{attribute addProperty BoxType "EK1122-0000-0018"}
{attribute addProperty Id "Beckhoff_EPP3xxxsub_EK1100EK1100_179A0949162A_0001_EPP3174_0002_0016EPP3174_B7B5302521026.25A_0002_EPP3174_0002_0017EPP3174_B7B5302521026.25A_0003_EPP3174_0002_0018EPP3174_B7B5302521026.25A_0004_EPP3184_0002_0016EPP3184_6082EBFD21026.25A_0005_EPP3184_0002_0017EPP3184_6082EBFD21026.25A_0006_EPP3184_0002_0018EPP3184_6082EBFD21026.25A_0007_EPP3184_0002_0019EPP3184_B7B5302521026.25A_0008_EPP3204_0002_0016EPP3204_72ABB95437847.25A_0009_EPP3204_0002_0017EPP3204_C91659E221026.25A_0010_EPP3204_0002_0018EPP3204_C91659E221026.25A_0011_EPP3204_0002_0019EPP3204_C91659E221026.25A_0012_EPP3314_0002_0016EPP3314_A69716D721026.25A_0013_EPP3314_0002_0017EPP3314_A69716D721026.25A_0014_EPP3314_0002_0018EPP3314_A69716D721026.25A_0015_EPP3632_0001_0016EPP3632_A724E07457872.25A_0016_EPP3632_0001_0017EPP3632_A724E07457872.25A_0017_EPP3744_0041_0016EPP3744_99A8040A38648.25A_0018_EPP3744_0041_0017EPP3744_99A8040A38648.25A_0019_EPP3744_0041_0018EPP3744_99A8040A38648.25A_0020_EPP3744_1041_0016EPP3744_99A8040A38648.25A_0021_EPP3744_1041_0017EPP3744_99A8040A38648.25A_0022_EPP3744_1041_0018EPP3744_99A8040A38648.25A_0023_EPP3744_1041_0019EPP3744_99A8040A38648.25A_0024_EPP3744_1041_0020EPP3744_99A8040A38648.25A_0025_EPP3752_0000_0017EPP3752_639ED5F327434.25"}
{attribute addProperty CRC "2472904185"}
{attribute addProperty SizeInBites "7642"}
{attribute addProperty SizeInBytes "955.25"}
TYPE Beckhoff_EPP3xxxEK1122_936585F9 EXTENDS EK1122_179A0949 :
STRUCT
	{attribute addProperty Name "Beckhoff_EPP3xxxsub_EK1100"}
	Beckhoff_EPP3xxxsub_EK1100 : EK1100_179A0949;
	{attribute addProperty Name "A_0001_EPP3174_0002_0016"}
	A_0001_EPP3174_0002_0016 : EPP3174_B7B53025;
	{attribute addProperty Name "A_0002_EPP3174_0002_0017"}
	A_0002_EPP3174_0002_0017 : EPP3174_B7B53025;
	{attribute addProperty Name "A_0003_EPP3174_0002_0018"}
	A_0003_EPP3174_0002_0018 : EPP3174_B7B53025;
	{attribute addProperty Name "A_0004_EPP3184_0002_0016"}
	A_0004_EPP3184_0002_0016 : EPP3184_6082EBFD;
	{attribute addProperty Name "A_0005_EPP3184_0002_0017"}
	A_0005_EPP3184_0002_0017 : EPP3184_6082EBFD;
	{attribute addProperty Name "A_0006_EPP3184_0002_0018"}
	A_0006_EPP3184_0002_0018 : EPP3184_6082EBFD;
	{attribute addProperty Name "A_0007_EPP3184_0002_0019"}
	A_0007_EPP3184_0002_0019 : EPP3184_B7B53025;
	{attribute addProperty Name "A_0008_EPP3204_0002_0016"}
	A_0008_EPP3204_0002_0016 : EPP3204_72ABB954;
	{attribute addProperty Name "A_0009_EPP3204_0002_0017"}
	A_0009_EPP3204_0002_0017 : EPP3204_C91659E2;
	{attribute addProperty Name "A_0010_EPP3204_0002_0018"}
	A_0010_EPP3204_0002_0018 : EPP3204_C91659E2;
	{attribute addProperty Name "A_0011_EPP3204_0002_0019"}
	A_0011_EPP3204_0002_0019 : EPP3204_C91659E2;
	{attribute addProperty Name "A_0012_EPP3314_0002_0016"}
	A_0012_EPP3314_0002_0016 : EPP3314_A69716D7;
	{attribute addProperty Name "A_0013_EPP3314_0002_0017"}
	A_0013_EPP3314_0002_0017 : EPP3314_A69716D7;
	{attribute addProperty Name "A_0014_EPP3314_0002_0018"}
	A_0014_EPP3314_0002_0018 : EPP3314_A69716D7;
	{attribute addProperty Name "A_0015_EPP3632_0001_0016"}
	A_0015_EPP3632_0001_0016 : EPP3632_A724E074;
	{attribute addProperty Name "A_0016_EPP3632_0001_0017"}
	A_0016_EPP3632_0001_0017 : EPP3632_A724E074;
	{attribute addProperty Name "A_0017_EPP3744_0041_0016"}
	A_0017_EPP3744_0041_0016 : EPP3744_99A8040A;
	{attribute addProperty Name "A_0018_EPP3744_0041_0017"}
	A_0018_EPP3744_0041_0017 : EPP3744_99A8040A;
	{attribute addProperty Name "A_0019_EPP3744_0041_0018"}
	A_0019_EPP3744_0041_0018 : EPP3744_99A8040A;
	{attribute addProperty Name "A_0020_EPP3744_1041_0016"}
	A_0020_EPP3744_1041_0016 : EPP3744_99A8040A;
	{attribute addProperty Name "A_0021_EPP3744_1041_0017"}
	A_0021_EPP3744_1041_0017 : EPP3744_99A8040A;
	{attribute addProperty Name "A_0022_EPP3744_1041_0018"}
	A_0022_EPP3744_1041_0018 : EPP3744_99A8040A;
	{attribute addProperty Name "A_0023_EPP3744_1041_0019"}
	A_0023_EPP3744_1041_0019 : EPP3744_99A8040A;
	{attribute addProperty Name "A_0024_EPP3744_1041_0020"}
	A_0024_EPP3744_1041_0020 : EPP3744_99A8040A;
	{attribute addProperty Name "A_0025_EPP3752_0000_0017"}
	A_0025_EPP3752_0000_0017 : EPP3752_639ED5F3;
END_STRUCT
END_TYPE

(* stored: Version 1.2.0.0, ProductVersion 3.1.4024.9
   DUT Beckhoff_EPP3xxxEK1122_936585F9: Id {0fc051ec-130c-45d1-8482-a521ddbd4362} *)
